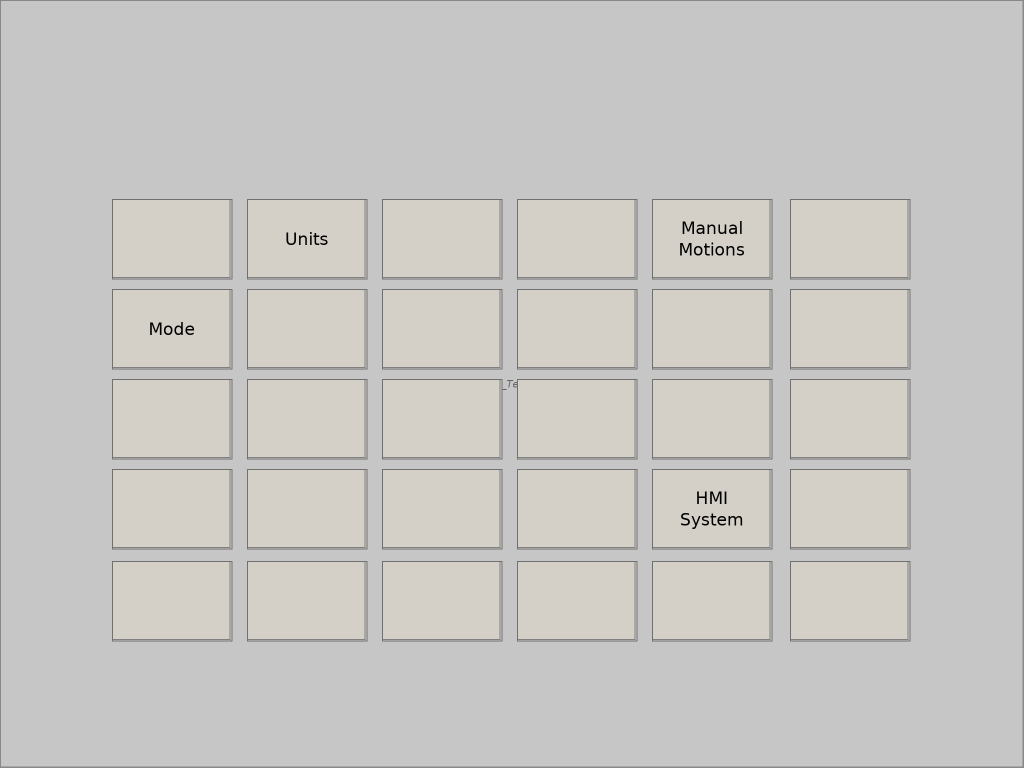
VISUALIZATION SS_10_MenuScreen  // 1024x768
    Frame (0,0 1024x768)
        shows SS_91_Template()
    Button (112,199 120x80), text list: ''
    Button (247,199 120x80), "Units", text list: ''
        OnMouseClick: change screen: Mc_01_Units
    Button (382,199 120x80), text list: ''
    Button (517,199 120x80), text list: ''
    Button (652,199 120x80), "Manual Motions", text list: ''
        OnMouseClick: change screen: SS_99_Motions
    Button (790,199 120x80), text list: ''
    Button (112,289 120x80), "Mode", text list: ''
        OnMouseClick: change screen: SS_01_ModeScreen
    Button (247,289 120x80), text list: ''
    Button (382,289 120x80), text list: ''
    Button (517,289 120x80), text list: ''
    Button (652,289 120x80), text list: ''
    Button (790,289 120x80), text list: ''
    Button (112,379 120x80), text list: ''
    Button (247,379 120x80), text list: ''
    Button (382,379 120x80), text list: ''
    Button (517,379 120x80), text list: ''
    Button (652,379 120x80), text list: ''
    Button (790,379 120x80), text list: ''
    Button (112,469 120x80), text list: ''
    Button (247,469 120x80), text list: ''
    Button (382,469 120x80), text list: ''
    Button (517,469 120x80), text list: ''
    Button (652,469 120x80), "HMI System", text list: ''
        OnMouseClick: change screen: SS_11_HMISystem
    Button (790,469 120x80), text list: ''
    Button (112,561 120x80), text list: ''
    Button (247,561 120x80), text list: ''
    Button (382,561 120x80), text list: ''
    Button (517,561 120x80), text list: ''
    Button (652,561 120x80), text list: ''
    Button (790,561 120x80), text list: ''
END_VISUALIZATION

(* stored: Version 1.1.0.1, ProductVersion 3.1.4024.12
   Visu SS_10_MenuScreen: Id {fcfc6bab-7c77-4a3a-b5c7-4b3a5f95aa3f} *)
